// TIA Portal V16 export
// export: Created 2024-09-05T17:39:22.0304242Z, ExportSetting WithDefaults, DisplayName Totally Integrated Automation Portal, DisplayVersion V16 Update 6, DisplayName TIA Portal Version Control Interface, DisplayVersion V16 Update 2, DisplayName TIA Portal Openness, DisplayVersion V16 Update 6, DisplayName STEP 7 Professional, DisplayVersion V16 Update 6, DisplayName STEP 7 Safety, DisplayVersion V16, DisplayName WinCC Advanced, DisplayVersion V16 Update 6
DATA_BLOCK "Main_Safety_RTG1_DB"   // DB48, F_DB
NAME : FUSI
VERSION : 0.1
// stored: AutoNumber true, DBAccessibleFromOPCUA true, InstanceOfName Main_Safety_RTG1, InstanceOfType FB
"Main_Safety_RTG1"
   // VAR
   //    ACK_GL_Instance : ACK_GL;
   //    "ESTOP1_3L+" : ESTOP1;
   //    "FDBACK_A2.7" : FDBACK;
   //    "ESTOP1_4L+" : ESTOP1;
   //    "FDBACK_A2.8" : FDBACK;
   //    "FDBACK_A2.9" : FDBACK;
   //    "ESTOP1_5L+" : ESTOP1;
   //    "F_IEC_Timer_3L+" : TON;
   //    "F_IEC_Timer_4L+" : TON;
   //    FDBACK_KF101x : FDBACK;
   //    FDBACK_KM20_KM21 : FDBACK;
   // END_VAR
BEGIN
END_DATA_BLOCK
